// TIA Portal V16 export
// export: Created 2022-01-12T14:34:29.9748451Z, ExportSetting WithDefaults, DisplayName Totally Integrated Automation Portal, DisplayVersion V16 Update 4, DisplayName TIA Portal Version Control Interface, DisplayVersion V16 Update 2, DisplayName TIA Portal Openness, DisplayVersion V16 Update 4, DisplayName STEP 7 Professional, DisplayVersion V16 Update 4, DisplayName STEP 7 Safety, DisplayVersion V16, DisplayName WinCC Professional, DisplayVersion V16 Update 4
TYPE "typFunkcjeObiektówCipu"
// stored: IsFailsafeCompliant false
   STRUCT
      "-na stacji CIP duże zbiorniki i zawory pod nimi" : Bool;   // tor0 to urządzenia wykorzystywane podczas pracy obu torów 1 i 2
      pompaPodawaniaCip : Int;   // najczęściej na torach 1 i 2
      zawórZrzutowyDoKanalizacji : Int;   // najczęściej na torach 1 i 2
      zawórWydawczyCip : Int;   // najczęściej na torach 1 i 2
      zawórBypassPrzygotowaniaStacji : Int;   // najczęściej na torach 1 i 2
      zawórParowyOdcinający : Int;   // najczęściej na torach 1 i 2
      zawórParowyRegulacyjny : Int;   // najczęściej na torach 1 i 2
      zawórWydawczyWodyWtórnej : Int;   // najczęściej na torach 1 i 2
      zawórPowrotnyWodyWtórnej : Int;   // najczęściej na torach 1 i 2
      zawórWydawczyŁugu : Int;   // najczęściej na torach 1 i 2
      zawórPowrotnyŁugu : Int;   // najczęściej na torach 1 i 2
      zawórWydawczyKwasu : Int;   // najczęściej na torach 1 i 2
      zawórPowrotnyKwasu : Int;   // najczęściej na torach 1 i 2
      zawórWydawczyWodyCzystej : Int;   // najczęściej na torach 1 i 2
      zawórWydawczyDezynfekantu : Int;   // najczęściej na torach 1 i 2 - patrz Orzeł2 2019_1109
      zawórWydawczyDezynfekantu_2 : Int;   // najczęściej na torach 1 i 2 - patrz Orzeł2 2019_1109
      zawórPowrotnyDezynfekantu : Int;   // najczęściej na torach 1 i 2 - patrz Orzeł2 2019_1109
      zawórPowrotnyDezynfekantu_2 : Int;   // najczęściej na torach 1 i 2 - patrz Orzeł2 2019_1109
      zawórStopowyPowrotuDezynfekantu : Int;   // najczęściej na torach 1 i 2 - patrz Orzeł2 2019_1109
      zawórStopowyPowrotuDezynfekantu_2 : Int;   // najczęściej na torach 1 i 2 - patrz Orzeł2 2019_1109
      zawórNaGruszkęZbiornikaŁugu : Int;   // najczęściej na torze 1 lub na torze 2 (mycie się stacji)
      zawórNaGruszkęZbiornikaKwasu : Int;   // najczęściej na torze 1 lub na torze 2 (mycie się stacji)
      zawórNaGruszkęZbiornikaWodyWtórnej : Int;   // najczęściej na torze 1 lub na torze 2 (mycie się stacji)
      zawórNaGruszkęZbiornikaWodyCzystej : Int;   // najczęściej na torze 1 lub na torze 2 (mycie się stacji)
      zawórNaGruszkęZbiornikaDezynfekantu : Int;   // najczęściej na torach 1 i 2 - patrz Orzeł2 2019_1109
      zawórNaGruszkęZbiornikaDezynfekantu_2 : Int;   // najczęściej na torach 1 i 2 - patrz Orzeł2 2019_1109
      zawórWodaNaGruszkęZbiornikaDezynfekantu_2 : Int;   // najczęściej na torach 1 i 2 - patrz Orzeł2 2019_1109
      zawórUzupełnianiaWodyCzystejZbŁugu : Int;   // najczęsciej tor 0
      zawórUzupełnianiaWodyCzystejZbKwasu : Int;   // najczęsciej tor 0
      zawórUzupełnianiaWodyCzystejZbWodyWtórnej : Int;   // najczęsciej tor 0
      zawórUzupełnianiaWodyCzystejZbWodyCzystej : Int;   // najczęsciej tor 0
      ZawórUzupełnianiaWodyCzystejZbDezynfekantu : Int;   // najczęsciej tor 0
      ZawórUzupełnianiaWodyCzystejZbDezynfekantu_2 : Int;   // najczęsciej tor 0
      "---zbiorniki główne na stacji CIP -czujniki" : Bool;
      zbiornikŁugu : Struct
         czujnikDolnegoPoziomu : Int;
         czujnikGórnegoPoziomu : Int;
         temperatura : Int;
         poziomAnalogowy : Int;
         czujnikwłazu : Int;
      END_STRUCT;
      zbiornikKwasu : Struct
         czujnikDolnegoPoziomu : Int;
         czujnikGórnegoPoziomu : Int;
         temperatura : Int;
         poziomAnalogowy : Int;
         czujnikwłazu : Int;
      END_STRUCT;
      zbiornikWodyWtórnej : Struct
         czujnikDolnegoPoziomu : Int;
         czujnikGórnegoPoziomu : Int;
         temperatura : Int;
         poziomAnalogowy : Int;
         czujnikwłazu : Int;
      END_STRUCT;
      zbiornikwodyCzystej : Struct
         czujnikDolnegoPoziomu : Int;
         czujnikGórnegoPoziomu : Int;
         temperatura : Int;
         poziomAnalogowy : Int;
         czujnikwłazu : Int;
      END_STRUCT;
      zbiornikDezynfekantu : Struct
         czujnikDolnegoPoziomu : Int;
         czujnikGórnegoPoziomu : Int;
         temperatura : Int;
         poziomAnalogowy : Int;
         czujnikwłazu : Int;
         zbiornikDezynfekantu : Struct
            czujnikDolnegoPoziomu : Int;
            czujnikGórnegoPoziomu : Int;
            temperatura : Int;
            poziomAnalogowy : Int;
            czujnikwłazu : Int;
         END_STRUCT;
      END_STRUCT;
      zbiornikDezynfekantu_2 : Struct
         czujnikDolnegoPoziomu : Int;
         czujnikGórnegoPoziomu : Int;
         temperatura : Int;
         poziomAnalogowy : Int;
         czujnikwłazu : Int;
      END_STRUCT;
      "-zbiorniki na stacji przygotowania chemii" : Bool;
      zbiorniczekDozowaniaŁugu : Struct   // na stacji przygotowania chemii
         czujnikDolnegoPoziomu : Int;
         czujnikGórnegoPoziomu : Int;
         temperatura : Int;
         poziomAnalogowy : Int;
         czujnikwłazu : Int;
         zbiornikDezynfekantu : Struct
            czujnikDolnegoPoziomu : Int;
            czujnikGórnegoPoziomu : Int;
            temperatura : Int;
            poziomAnalogowy : Int;
            czujnikwłazu : Int;
         END_STRUCT;
      END_STRUCT;
      zbiorniczekDozowaniaKwasu : Struct   // na stacji przygotowania chemii
         czujnikDolnegoPoziomu : Int;
         czujnikGórnegoPoziomu : Int;
         temperatura : Int;
         poziomAnalogowy : Int;
         czujnikwłazu : Int;
         zbiornikDezynfekantu : Struct
            czujnikDolnegoPoziomu : Int;
            czujnikGórnegoPoziomu : Int;
            temperatura : Int;
            poziomAnalogowy : Int;
            czujnikwłazu : Int;
         END_STRUCT;
      END_STRUCT;
      zbiorniczekDozowanieDezynfekantu : Struct   // na stacji przygotowania chemii
         czujnikDolnegoPoziomu : Int;
         czujnikGórnegoPoziomu : Int;
         temperatura : Int;
         poziomAnalogowy : Int;
         czujnikwłazu : Int;
         zbiornikDezynfekantu : Struct
            czujnikDolnegoPoziomu : Int;
            czujnikGórnegoPoziomu : Int;
            temperatura : Int;
            poziomAnalogowy : Int;
            czujnikwłazu : Int;
         END_STRUCT;
      END_STRUCT;
      "--nalinii" : Bool;
      temperaturaZaWymiennikiem : Int;   // najczęściej na torach 1 i 2
      przepływomierzZaWymiennikiem : Int;   // najczęściej na torach 1 i 2
      temperaturaNaPowrocie : Int;   // najczęściej na torach 1 i 2
      przewodnośćNaPowrocie : Int;   // najczęściej na torach 1 i 2
      czujnikPrzepływuNaPowrocie : Int;   // najczęściej na torach 1 i 2
      "-naobiekcie" : Bool;
      czujnikDolnegoPoziomuwZbiornikuDrenowanym : Int;   // najczęściej na torach 1 i 2 (sygnał z obiektu mytego)
      "-przygotowaniechemii" : Bool;
      pompkaDozowaniaŁuguwLinię : Int;   // najczęsciej tor 0
      pompkaDozowaniaKwasuwLinię : Int;   // najczęsciej tor 0
      pompkaDozowaniaDezynfekantuwLinię : Int;   // najczęściej na torach 1 i 2
      zawórDozowaniaLuguwLinię : Int;   // najczęściej na torach 1 i 2
      zawórDozowaniaKwasuwLinię : Int;   // najczęściej na torach 1 i 2
      zawórDozowaniaDezynfekantuwLinię : Int;   // najczęściej na torach 1 i 2
      czujnikPrzepływuDozowanegoŁugu : Int;   // najczęsciej tor 0
      czujnikPrzepływuDozowanegoKwasu : Int;   // najczęsciej tor 0
      czujnikPrzepływuDozowanegoDezynfekantu : Int;   // najczęściej na torach 1 i 2
      PrzepływomierzDozowanejChemii : Int;   // najczęsciej tor 0
   END_STRUCT;
END_TYPE
